PROGRAM prgPV
VAR
	fbPV						: FB_Hoymiles_DTU_ProS_PV_Inverter;
	fbEnphase					: FB_Enphase;
	fbPVCounter					: FB_EnergyCounter;
	lrPowerPVEnphase_W			: LREAL;
	lrPowerPV					: LREAL;						//{#lynus.ag#()}
	byErrorWarningPV			: BYTE;							//{#lynus.ag#()}
END_VAR
VAR PERSISTENT
	lrCounterPV					: LREAL;						//{#lynus.ag#()}
	bEnable						: BOOL;
	str_IP						: STRING(15);
END_VAR

// To-Do:
// adopt FB Declaration, change to correct FB
// adopt FB Definition, change to correct in/out Vars
// correct lrPowerPV definition
// correct lrCounterPV definition
// correct byErrorWarningPV definition


// PV config for external Inverter

(*
fbPV(
	bEnable:= bEnable, 
	sIPAdress:= str_IP, 
	byUnitID_Inverter:= 1, 
	stDataEMPower_PV=> , 
	stDataEMCounter_PV=> , 
	diNrOfEM_OUT_PV=> );
// operation state of the inverter is unclear if that is ok, no documentation from Hoymiles

lrPowerPV := fbPV.DataHoymiles_DTU_Pro_Total.lrPowerAcInverter;
byErrorWarningPV := fbPV.stDataEMPower_PV.byErrorWarning;

IF fbPV.stDataEMCounter_PV.lrCounterEnergyT1_Production > lrCounterPV THEN  	
	lrCounterPV := fbPV.stDataEMCounter_PV.lrCounterEnergyT1_Production;
END_IF

*)


// PV config for Enphase Gateway

fbEnphase(
	bStart:= TRUE, 
	tDelayRequest:= T#3S, 
	sHostname:= '192.168.1.30', 
	bValidResult=> , 
	bBusy=> , 
	bError=> , 
	bDone=> , 
	hrErrorCode=> ,
	lrpowerprod => lrPowerPVEnphase_W );
	
// re-calc Power to kW
lrPowerPV := lrPowerPVEnphase_W / 1000;

fbPVCounter(
	byActiveTariff:= 1, 
	lrPowerInput:= lrPowerPV, 
	lrTotalCounterEnergy_Consumption=> , 
	lrTotalCounterEnergy_Production=> , 
	lrCounterEnergyT1_Consumption=> , 
	lrCounterEnergyT2_Consumption=> , 
	lrCounterEnergyT1_Production=> , 
	lrCounterEnergyT2_Production=> );
	
IF fbPVCounter.lrTotalCounterEnergy_Consumption > lrCounterPV THEN  	
	lrCounterPV := fbPVCounter.lrTotalCounterEnergy_Consumption;
END_IF

END_PROGRAM

(* stored: Version 1.1.0.1, ProductVersion 3.1.4024.11
   POU prgPV: Id {52a4cf08-62d2-4b94-900b-2ea0759cae15}, SpecialFunc None *)
